// Mitsubishi GX Works2 project: 东芝分拣通信   PLC: Q10UDEH

TYPE ConveyorIO : STRUCT
  xUnloadCCW : BOOL;  (* 下料为反转 *)
  xUnloadAlarm : BOOL;  (* 下料报警 *)
  xUnload : BOOL;  (* 下料请求 *)
  xPutInto : BOOL;  (* 线体直接投入物料 *)
  xNotArriveAlarm : BOOL;  (* 未到达报警 *)
  xNextRun : BOOL;  (* 下段线体运行 *)
  xMotorCW : BOOL;  (* 电机正转 *)
  xMotorCCW : BOOL;  (* 电机反转 *)
  xManual : BOOL;  (* 手动 *)
  xloadCCW : BOOL;  (* 上料为反转 *)
  xLimitAlarrm : BOOL;  (* 限位报警 *)
  xLoad : BOOL;  (* 上料请求 *)
  xForward : BOOL;  (* 正转手动 *)
  xEmpty : BOOL;  (* 线体状态为空 *)
  xCWPresent : BOOL;  (* 正转检测有无传感器 *)
  xCCWPresent : BOOL;  (* 反转检测有无传感器 *)
  xBusy : BOOL;  (* 工作中 *)
  xBackward : BOOL;  (* 反转手动 *)
  xAuto : BOOL;  (* 自动 *)
  xPosLimit : BOOL;  (* 正限位 *)
  xNegLimit : BOOL;  (* 负限位 *)
  xOverWidthAlarm : BOOL;  (* 超宽报警 *)
  xError : BOOL;  (* 报警 *)
  iProductCategoryIn : INT;  (* 产品类型输入 *)
  iProductCategory : INT;  (* 产品类型记录 *)
  iProductCategoryOut : INT;  (* 产品类型输出 *)
  diDeviceID : DINT;  (* 设备编号 *)
  tUnloadAlarmDelay : TIME;  (* 下料报警时间设置 *)
  tLoadDelay : TIME;  (* 上料延时设置 *)
  xSizeDeficientDetect : BOOL;  (* 尺寸缺陷检测 *)
  xZoneClear : BOOL;  (* 初始化线体清除 *)
  tZoneClearTime : TIME;  (* 初始化线体清除时间 *)
  iTaskIDIn : INT;  (* 产品类型输入 *)
  iTaskID : INT;  (* 产品类型记录 *)
  iTaskIDOut : INT;  (* 产品类型输出 *)
  diDesConveyorIn : DINT;  (* 产品类型输入 *)
  diDesConveyor : DINT;  (* 产品类型记录 *)
  diDesConveyorOut : DINT;  (* 产品类型输出 *)
END_STRUCT END_TYPE

TYPE FanucRobotIO : STRUCT
  o_xColumn : ARRAY [0..3] OF BOOL;  (* 行号 *)
  o_xRow : ARRAY [0..3] OF BOOL;  (* 列号 *)
  o_xPutNumber : ARRAY [0..3] OF BOOL;  (* 放料位 *)
  o_xSortStart : BOOL;  (* 开始启动 *)
  i_xPutOver : BOOL;  (* 放货完成 *)
  i_xPickOver : BOOL;  (* 取货完成 *)
END_STRUCT END_TYPE

TYPE SortCommunicationIO : STRUCT
  i_iResponsPCPLC : INT;  (* 上位机写入-应答 *)
  i_iSortDoneAknPCPLC : INT;  (* 上位机写入-任务处理完成 *)
  i_arriBatteryStatus : ARRAY [1..128] OF INT;  (* 上位机写入-电池状态 *)
  o_iRequestPLCPC : INT;  (* 上位机读取-请求 *)
  o_iSortDonePLCPC : INT;  (* 上位机读取-分拣完成 *)
  i_iInfoWriteDone : INT;  (* 上位机写入-参数写入完成 *)
  i_xSortOver : BOOL;  (* 按钮，分拣完成 *)
  o_xSortDone : BOOL;  (* 状态，分拣完成 *)
END_STRUCT END_TYPE

// global labels: Global
VAR_GLOBAL
  g_xAuto AT M11 : BOOL;
  g_xManual : BOOL;
  g_xEStop AT X0 : BOOL;
  g_xReset : BOOL;
  g_xStackLampRed AT Y200 : BOOL;  (* 塔灯红 *)
  g_xStackLampAmber AT Y201 : BOOL;  (* 塔灯黄 *)
  g_xStackLampGreen AT Y202 : BOOL;  (* 塔灯绿 *)
  g_xBuzzer AT Y203 : BOOL;  (* 蜂鸣器 *)
  g_xStop AT X3 : BOOL;
  g_xAutoStart AT X2 : BOOL;  (* 启动按钮 *)
  g_xRemoteAutoStart AT M0 : BOOL;
  g_xRemoteAuto AT M10 : BOOL;
  g_iState AT D40 : INT;  (* 状态显示 *)
  g_iLocalAutoStep : BOOL;
  g_xAlarm : BOOL;
  g_xPause AT M3 : BOOL;  (* 暂停 *)
  g_diDeviceIDSelect AT D0 : DINT;
  g_xResetSingle AT M4 : BOOL;  (* 单线体复位 *)
  g_xInsertTask AT M5 : BOOL;  (* 插入任务 *)
  g_iInsertTaskID AT D2 : INT;  (* 插入任务号 *)
  g_iConveyorStatus AT D4 : INT;
  g_iInsertCategory AT D6 : INT;
  g_diInsertDesConveyor AT D8 : DINT;
  g_x20TcpFailed : BOOL;  (* 30预20通讯失败 *)
  g_xAutoLamp AT Y204 : BOOL;  (* 启动灯 *)
  g_iLoadTask AT D50 : ARRAY [0..13] OF INT;  (* 排队任务站，D50-D62 *)
  g_xAutoSwitch AT X1 : BOOL;  (* 手自动钥匙旋钮 *)
  g_xMute AT M2 : BOOL;  (* 静音按钮，报警消除时复位 *)
  g_xResetTask1 AT M9 : BOOL;  (* 复位排队任务按钮 *)
  g_xLoadPermit : ARRAY [1..2] OF BOOL;  (* 定位机排队任务允许 *)
  g_x40TcpFailed : BOOL;  (* 30预40通讯失败 *)
  g_xForceImport AT M1 : BOOL;  (* 强制入库 *)
  g_x24HourImport1Forbidden AT M12 : BOOL;  (* 24小时入库禁止1 *)
  g_x24HourImport2Forbidden AT M13 : BOOL;  (* 24小时入库禁止2 *)
  g_xPreChemImport1Forbidden AT M14 : BOOL;  (* 预化成入库禁止1 *)
  g_xPreChemImport2Forbidden AT M15 : BOOL;  (* 预化成入库禁止2 *)
  g_x24HourExport1Forbidden AT M16 : BOOL;  (* 24小时出库禁止 *)
  g_xPreChemExport1Forbidden AT M17 : BOOL;  (* 预化成出库禁止1 *)
  g_xPreChemExport2Forbidden AT M18 : BOOL;  (* 预化成出库禁止2 *)
  g_xPickDone : BOOL;  (* 分拣完成 *)
  g_xPickOver AT X4 : BOOL;  (* 注液机给我们的信号，待定 *)
END_VAR

// task Task_01 (event TRUE, interval 0, priority 31): POU_01

PROGRAM POU_01
VAR
  SortCommunication70210 : SortCommunication;  (* 分拣通信 *)
  Conveyor70210 : Conveyor;  (* 分拣线体 *)
  ConveyorIO70210 : ConveyorIO;  (* 分拣线体 *)
  RobotIO70210 : FanucRobotIO;  (* 分拣机器人 *)
  SortCommunicationIO70210 : SortCommunicationIO;  (* 分拣通信 *)
  ConveyorIO70211 : ConveyorIO;  (* 分拣线体的下一段线体，举个例子 *)
END_VAR
Conveyor70210(ConveyorMotor:=ConveyorIO70210);

SortCommunication70210(ConveyorIO:=ConveyorIO70210,SortCommunicationIO:= SortCommunicationIO70210 ,FanucRobotIO:= RobotIO70210);
SortCommunicationIO70210 .i_iResponsPCPLC:=D2705;
SortCommunicationIO70210 .i_iInfoWriteDone:=D2706;
SortCommunicationIO70210 .i_iSortDoneAknPCPLC:=D2707;
D3705:=SortCommunicationIO70210 .o_iRequestPLCPC;(*有料请求*)
D3706:=SortCommunicationIO70210 .o_iSortDonePLCPC;(*分拣完成信号*)
FOR Z0:=0 TO 127 BY 1 DO
	SortCommunicationIO70210 .i_arriBatteryStatus[Z0+1]:=D2708Z0;
END_FOR;

SortCommunicationIO70210.i_xSortOver:=X2;(*这个是手动放行按钮，可要可不要*)
RobotIO70210.i_xPickOver:=X0;(*机器人给的取货完成*)
RobotIO70210.i_xPutOver:=X1;(*机器人给的放货完成*)
Y0:=RobotIO70210.o_xSortStart;(*给机器人的开始启动*)
Y1:=RobotIO70210.o_xColumn[0];(*给机器人的行号*)
Y2:=RobotIO70210.o_xColumn[1];
Y3:=RobotIO70210.o_xColumn[2];
Y4:=RobotIO70210.o_xColumn[3];
Y5:=RobotIO70210.o_xRow[0];(*给机器人的列号*)
Y6:=RobotIO70210.o_xRow[1];
Y7:=RobotIO70210.o_xRow[2];
Y8:=RobotIO70210.o_xRow[3];
Y9:=RobotIO70210.o_xPutNumber[0];(*给机器人的放料位置*)
YA:=RobotIO70210.o_xPutNumber[1];
YB:=RobotIO70210.o_xPutNumber[2];
YC:=RobotIO70210.o_xPutNumber[3];

ConveyorIO70210.xUnload:=SortCommunicationIO70210.o_xSortDone AND ConveyorIO70211.xEmpty;(*比普通的下料多了个判断条件，需要分拣完成再下料*)
END_PROGRAM

FUNCTION_BLOCK SortCommunication
VAR
  m_iStep : INT;
END_VAR
VAR_IN_OUT
  ConveyorIO : ConveyorIO;
  SortCommunicationIO : SortCommunicationIO;
END_VAR
VAR
  m_iCoordinateX : INT;
  m_iCoordinateY : INT;
END_VAR
VAR_IN_OUT
  FanucRobotIO : FanucRobotIO;
END_VAR
VAR_OUTPUT
  o_iErrorNub : INT;
END_VAR
VAR
  ii : INT;
END_VAR
VAR CONSTANT
  ROW_NUB : INT := 8;  (* 每排的数量 *)
END_VAR
VAR
  m_xEno : BOOL;
END_VAR
(*********************************************************)
(*
DB1区(PC->PLC)100个字		
"字(16位）序号
(从1开始)"	功能描述	具体参数解释
1	应答	"1：复位
2：读码成功(参数写入完成)
101：条码空
102：条码规则校验失败
103：步号校验失败"
2	任务处理完成	"1：复位
2：处理完成"
3	"电芯状态，
128个电芯"	一个字代表两个电芯状态，1：合格，2,3,4:NG 

DB2区(PLC->PC)10个字		
"字(16位）序号
(从1开始)"	功能描述	具体参数解释
请求	"1：无板
2：请求分拣
"
分拣完成	"1：复位
2：挑选完成
3：撤销
"
跟机器人通信13个输出，2个输入
						13个输出分别是：4个表示行，4个表示列，4个表示不良信息，1个启动信号
						2个输入分别是：抓料完成，放料完成		

*)
(*********************************************************)
IF g_xAuto THEN
	(*——这里临时改一下，暂时人工挑选,所以需要分拣完成按钮——*)	
		IF LDP(TRUE,SortCommunicationIO.i_xSortOver)THEN
			m_iStep:=4;
		END_IF;(**)
(*——以上是暂时人工分拣的，以后删掉——*)
	CASE m_iStep OF
		0:(*//初始化*)
		SortCommunicationIO.o_iRequestPLCPC:=1;
		SortCommunicationIO.o_iSortDonePLCPC:=1;
		ii:=0;
		SortCommunicationIO.o_xSortDone:=0;
		m_iStep:=1;
		
		1:(*发送框码的扫码请求*)
		IF ConveyorIO.xEmpty THEN
			SortCommunicationIO.o_iRequestPLCPC:=1;
		ELSE
			SortCommunicationIO.o_iRequestPLCPC:=2;(*发2表示有料了，他就会扫码*)
		END_IF;
		(*//请求确认*)
		IF SortCommunicationIO.o_iRequestPLCPC=2 THEN(*加个条件，免得无脑跳Step2*)
			CASE SortCommunicationIO.i_iResponsPCPLC OF 
			0:;
			1:;(*//复位*)
			2:(*//读码（入库申请）成功*)
				m_iStep:=2;
				ii:=0;
				m_iCoordinateX:=1;(*//框码扫码成功后把坐标改为1,1*)
				m_iCoordinateY:=1;
			3:(*//取放货完成*)
				ConveyorIO.xPutInto:=1; 
			4:(*//旋转*)
				;
			5:(*//不旋转*)
				;
			101:(*//条码空*)
				o_iErrorNub:=101;
			102:(*//条码规则检验失败*)
				o_iErrorNub:=102;
			103:(*//步号校验失败*)
				o_iErrorNub:=103;
			104:(*//无库位可用*)
				o_iErrorNub:=104;
			END_CASE;
		END_IF;	
		
		2:(*//料框位置抓取*)		
		IF ii=129 THEN(*129表示所有有问题的都抓完了*)
			m_iStep:=4;
		ELSE(*有不良品*)
			FanucRobotIO.o_xSortStart:=1;(*//从料框取料*)
			FanucRobotIO.o_xColumn[3]:=m_iCoordinateX/8=1;(*XY的偏移量计算在末尾*)
			FanucRobotIO.o_xColumn[2]:=(m_iCoordinateX MOD 8)/4=1;
			FanucRobotIO.o_xColumn[1]:=(m_iCoordinateX MOD 4)/2=1;
			FanucRobotIO.o_xColumn[0]:=(m_iCoordinateX MOD 2)/1=1;
			FanucRobotIO.o_xRow[3]:=m_iCoordinateY/8=1;			
			FanucRobotIO.o_xRow[2]:=(m_iCoordinateY MOD 8)/4=1;
			FanucRobotIO.o_xRow[1]:=(m_iCoordinateY MOD 4)/2=1;
			FanucRobotIO.o_xRow[0]:=(m_iCoordinateY MOD 2)/1=1;
			CASE SortCommunicationIO.i_arriBatteryStatus[ii] OF
			1:(*合格*)
					;
			2:(*容量不足*)
					FanucRobotIO.o_xPutNumber[0]:=1;	
			3:(*电压不足*)
					FanucRobotIO.o_xPutNumber[1]:=1;	
			4:(*阻值错误*)
					FanucRobotIO.o_xPutNumber[2]:=1;	
			5:(*电压过高*)
					FanucRobotIO.o_xPutNumber[3]:=1;	
			END_CASE;
		END_IF;
		IF LDP(TRUE,FanucRobotIO.i_xPickOver) THEN(*//抓取动作完成*)
			m_iStep:=3;
		END_IF;
	
		3:(*//放入下料皮带线*)
			FanucRobotIO.o_xSortStart:=0;(*//从料框取料*)
			FanucRobotIO.o_xColumn[3]:=0;(*XY的偏移量计算在末尾*)
			FanucRobotIO.o_xColumn[2]:=0;
			FanucRobotIO.o_xColumn[1]:=0;
			FanucRobotIO.o_xColumn[0]:=0;
			FanucRobotIO.o_xRow[3]:=0;
			FanucRobotIO.o_xRow[2]:=0;
			FanucRobotIO.o_xRow[1]:=0;
			FanucRobotIO.o_xRow[0]:=0;
		IF LDP(TRUE,FanucRobotIO.i_xPutOver) THEN(*//抓取动作完成*)
		(*这个得放货完成在复位，方便step2给*)
		FanucRobotIO.o_xPutNumber[0]:=0;
		FanucRobotIO.o_xPutNumber[1]:=0;
		FanucRobotIO.o_xPutNumber[2]:=0;
		FanucRobotIO.o_xPutNumber[3]:=0;
			m_iStep:=2;
		END_IF;	
		
		4:
		IF  NOT SortCommunicationIO.o_xSortDone  THEN(*这里表示只给一下2*)
				SortCommunicationIO.o_iSortDonePLCPC:=2;
				SortCommunicationIO.o_xSortDone:=1;
		END_IF;		
		IF SortCommunicationIO.i_iSortDoneAknPCPLC =2 THEN
			SortCommunicationIO.o_iSortDonePLCPC:=1;
			m_iCoordinateX:=1;
			m_iCoordinateY:=1;
		END_IF;	
			IF ConveyorIO.xEmpty THEN
				m_iStep:=0;
			END_IF;
	END_CASE;
	IF LDP(TRUE,m_iStep=2 AND SortCommunicationIO.i_iInfoWriteDone=2) THEN(*判断哪个地方是有问题的*)
		FOR ii:=ii+1 TO 128 BY 1 DO
			IF SortCommunicationIO.i_arriBatteryStatus[ii]<>1 THEN
				m_iCoordinateX:=((ii-1) MOD ROW_NUB);
				m_iCoordinateY:=(ii-1)/ROW_NUB+1;(*把上位机给的编号值对应到二维的偏移上*)
				EXIT;
			END_IF;
		END_FOR;
	END_IF;
END_IF;(*g_xauto*)	
IF  g_diDeviceIDSelect=ConveyorIO.diDeviceID AND g_xResetSingle THEN(*复位线体时，同时复位步数和请求，重新来一遍*)
	m_iStep:=0;
END_IF;	
IF  NOT g_xAuto THEN
		SortCommunicationIO.o_iRequestPLCPC:=0;
		SortCommunicationIO.o_iSortDonePLCPC:=0;
END_IF;
END_FUNCTION_BLOCK

FUNCTION_BLOCK Conveyor
VAR
  m_xPresentDelay : BOOL;  (* 有无判断延时 *)
  m_xLoadDelayOut : BOOL;  (* 上料延时输出 *)
  m_xInitial : BOOL;  (* 初始化 *)
  m_tUnloadTimer : TIME;  (* 下料计时器 *)
  m_tPresentDelayCurrentTime : TIME;
  m_tonUnloadAlam : TON;  (* 下料报警定时器 *)
  m_tonPresentDelay : TON;  (* 物料有无判断延时，防止误动作 *)
  m_tonNotArriveAlarm : TON;  (* 未到达报警计时 *)
  m_tonLoadDelay : TON;  (* 上料延时 *)
  m_tNotArriveCurrentTime : TIME;  (* 未到达报警计时当前时间 *)
  m_tLoadTimer : TIME;  (* 上料计时器 *)
  iStep : INT;  (* 上料步骤 *)
  m_wStateWord : INT;
END_VAR
VAR_IN_OUT
  ConveyorMotor : ConveyorIO;  (* 输送线输入输出 *)
END_VAR
VAR
  m_tonZoneClear : TON;  (* 初始化清除 *)
  m_tZoneClearCurrentTime : TIME;  (* 初始化清除当前时间 *)
  m_xAutoClear : BOOL;  (* 初始化清除标志位 *)
  m_xZoneClearDone : BOOL;  (* 初始化清除完成 *)
END_VAR
(*////////////////////////////////////////////////////////////////////////////////////////////////////////////
//传输线控制FB块，可控制单方向线体，双向旋转线体，支持双向上下料            
//线体初始化后为空的情况下输入xLoad信号即可进行上料动作，使用xLoadCCW信号可反方向上料
//增加了产品信息和产品种类的储存，当传输线为空和上料进行标志位为零的情况下清除产品信息和产品种类
//使用方式是在置位xLoad信号后，把产品信息和产品种类传入，等下料后自动清零
//线体不为空的情况下使用xUnload信号可进行下料动作，物料有无传感器的下降沿后出发计时器，延时断开传输线旋转
//单方向传输线体把xLoadCCW、xUnloadCCW设置为零，双向线体上料方向和下料反向的,方向固定的 把xUnloadCCW设置为1
//双方向线体双向都能上下料的要根据上料的方向来设置xLoadCCW,xUnloadCCW
//增加工作中信号xBusy当电机正转 显示为工作中
//增加上下料超时报警，xLoadAlarm，xUnloadAlarm，设定时间在LOAD_UNLOAD_TIME常量上，现在设置的为30秒
//增加xPutInto信号，用于直接投入的物料，检测开关感应到后，直接进入下料流程，上升沿有效
//离开延时改为变量 iLeaveDelay 默认为0 离开检测开关离输送线尾端比较远的线体需要根据情况设定100ms为单位
//增加初始化标志位，增加进入延时时间，初始化为进入延时时间为0 ，离开延时时间为2S，通过外围接口可以更改
//修改信息  修改后请增加版本
//12-17进行了优化，增加了未到达报警，当物料未传送到下一设备，就报未到达报警，使用xNextRun标志位制作，没有正常到达
//第0步，不能跳转到第一步把标志位复位，即出现中断情况，2秒后报警
//修改信息  修改后请增加版本
//上料延时增加为50ms防止干扰信号
//nextrun信号在 第三步也要复位
//增加限位报警
//增加超宽报警
//增加产品型号输出在下料的时候把产品型号输送给下一段线体
//增加线体单独复位
//增加任务插入功能配合全局变量
//增加暂停功能
//增加线体状态字显示  0 空闲 1：有料  2 工作中  3  超限报警 4 超宽报警  5 未到达报警  6 下料超时报警
//空料判断放在自动前，进行有无报警判断，然后跳转
//修改超限报警，与尺寸检测报警
////YAO      V1.0
//把所有的IF语句去掉，  IF语句占用指针存储区，容易造成存储区不足的现象
////YAO      V1.1
//初始化清除线体标志位xZoneClear
//ZPA zero pressure accumulation  Term that describes the Conveyor controls and mechanical scheme that will 
//cause loads to queue on a conveyor in discrete zones such that loads do not touch each other(wrapped boxed tray tote carton)
//除了产品信息外，还增加了目标地址，任务类型的数据传递。
//YAO      V1.0
///////////////////////////////////////////////////////////////////////////////////////////////////////////
(*********************************************************)
(*//初始化，
//上料延时位0S，下料报警延时为30S
//下料延时设一个比较大的时间，主要依靠xunload标志位来停止输送线，特殊情况可以用延时来停止物流线下料
//设置时间大的时候计时器会失效*)
IF NOT m_xInitial THEN
	ConveyorMotor.tLoadDelay:=T#100ms;
	ConveyorMotor.tUnloadAlarmDelay:=T#30s;
	ConveyorMotor.xPosLimit:=1;
	ConveyorMotor.xNegLimit:=1;
	ConveyorMotor.xSizeDeficientDetect:=0;
	ConveyorMotor.xZoneClear:=0;
	ConveyorMotor.tZoneClearTime:=T#10s;
	m_xInitial:=1;
END_IF;
(*//自动
//复位信号把步号置0，但xLoad与xUnload没有复位，调用程序需要注意复位后把这两个信号置零，以免发生误动作
//物料有无判断增加延时，防止开自动瞬间误动作发生*)
m_tonPresentDelay(IN:= ConveyorMotor.xCWPresent OR ConveyorMotor.xCCWPresent,
					PT:=T#100ms,
					Q:= m_xPresentDelay,
					ET:= m_tPresentDelayCurrentTime);
CASE iStep OF
0:(*//初始化*)
	ConveyorMotor.xMotorCW:=0;
	ConveyorMotor.xMotorCCW:=0;
	ConveyorMotor.xNextRun:=0;
	ConveyorMotor.iProductCategoryOut:=0;
	ConveyorMotor.iTaskIDOut:=0;
	ConveyorMotor.diDesConveyorOut:=0;
	out(NOT m_xPresentDelay,ConveyorMotor.xEmpty);(*	//判断物料有无传感器*)	
	mov(m_xPresentDelay AND g_xAuto AND NOT ConveyorMotor.xError,3,iStep);(*//自动情况下进行跳转*)(*无超限报警*)
	mov(NOT m_xPresentDelay AND g_xAuto AND NOT ConveyorMotor.xError,1,iStep);
1: (*//上料*)
	rst(ConveyorMotor.xLoad ,ConveyorMotor.iProductCategory);(*//上料开始清除产品信息*)
	rst(ConveyorMotor.xLoad ,ConveyorMotor.iTaskID);
	rst(ConveyorMotor.xLoad ,ConveyorMotor.diDesConveyor);
	mov(ConveyorMotor.xLoad,2,iStep);
2: (*//上料完成*)
	ConveyorMotor.iProductCategory:=ConveyorMotor.iProductCategoryIn;(* //产品信息传入*)
	ConveyorMotor.iTaskID:=ConveyorMotor.iTaskIDIn;
	ConveyorMotor.diDesConveyor:=ConveyorMotor.diDesConveyorIn;
	set(ConveyorMotor.xloadCCW,ConveyorMotor.xMotorCCW);
	rst(ConveyorMotor.xloadCCW,ConveyorMotor.xMotorCW);
	set(NOT ConveyorMotor.xloadCCW,ConveyorMotor.xMotorCW);
	rst(NOT ConveyorMotor.xloadCCW,ConveyorMotor.xMotorCCW);	
	m_tonLoadDelay(IN:= (ConveyorMotor.xCWPresent AND NOT ConveyorMotor.xloadCCW) 
												OR (ConveyorMotor.xCCWPresent AND ConveyorMotor.xloadCCW) ,
										PT:= ConveyorMotor.tLoadDelay ,
										Q:= m_xLoadDelayOut ,
										ET:= m_tLoadTimer );
	mov(m_xLoadDelayOut,3, iStep);
3:(*//下料请求*)	
	ConveyorMotor.xMotorCW:=0;
	ConveyorMotor.xMotorCCW:=0;
	ConveyorMotor.xEmpty:=0;
	mov(ConveyorMotor.xUnload AND NOT ConveyorMotor.xOverWidthAlarm,4,iStep);
4:(*	//下料完成*)
	set(ConveyorMotor.xUnloadCCW,ConveyorMotor.xMotorCCW);
	rst(ConveyorMotor.xUnloadCCW,ConveyorMotor.xMotorCW);
	set(NOT ConveyorMotor.xUnloadCCW,ConveyorMotor.xMotorCW);
	rst(NOT ConveyorMotor.xUnloadCCW,ConveyorMotor.xMotorCCW);	
	ConveyorMotor.xNextRun:=1; (*下一段线体旋转*)
	ConveyorMotor.iProductCategoryOut:=ConveyorMotor.iProductCategory;(*产品型号输出给下一段线体*)
	ConveyorMotor.iTaskIDOut:=ConveyorMotor.iTaskID;
	ConveyorMotor.diDesConveyorOut:=ConveyorMotor.diDesConveyor;
	mov( NOT ConveyorMotor.xUnload , 0, istep );
END_CASE;
(*In-feed zone clear and ready to accept a load from Upstream Conveyor*)
set(ldp(TRUE,g_xAuto) ,m_xAutoClear);
rst(ldf(TRUE,g_xAuto) ,m_xAutoClear);
m_tonZoneClear(IN:= m_xAutoClear AND ConveyorMotor.xZoneClear ,PT:= ConveyorMotor.tZoneClearTime ,Q:=m_xZoneClearDone ,ET:= m_tZoneClearCurrentTime );
set(m_xAutoClear AND ConveyorMotor.xZoneClear,ConveyorMotor.xMotorCW);
mov( m_xAutoClear AND ConveyorMotor.xZoneClear, 0 ,iStep );
rst(  ldf(TRUE, m_xAutoClear ) ,ConveyorMotor.xMotorCW);
rst( m_xZoneClearDone OR m_xPresentDelay  , m_xAutoClear );
(*投入上料，搬出下料，也可用来初始化*)
movp( ConveyorMotor.xPutInto, 0 , iStep );
(*//当前任务显示*)
movp( ConveyorMotor.diDeviceID=g_diDeviceIDSelect , ConveyorMotor.iProductCategory , g_iInsertCategory );
movp( ConveyorMotor.diDeviceID=g_diDeviceIDSelect , ConveyorMotor.iTaskID , g_iInsertTaskID );
dmovp( ConveyorMotor.diDeviceID=g_diDeviceIDSelect , ConveyorMotor.diDesConveyor , g_diInsertDesConveyor );
(*//插入任务*)
mov(g_xInsertTask AND ConveyorMotor.diDeviceID=g_diDeviceIDSelect ,g_iInsertCategory , ConveyorMotor.iProductCategory );
mov(g_xInsertTask AND ConveyorMotor.diDeviceID=g_diDeviceIDSelect , g_iInsertTaskID , ConveyorMotor.iTaskID );
dmov(g_xInsertTask AND ConveyorMotor.diDeviceID=g_diDeviceIDSelect , g_diInsertDesConveyor , ConveyorMotor.diDesConveyor );
(*//单线体复位，当设备号与本线体一致的时候执行复位*)
mov(g_xResetSingle AND ConveyorMotor.diDeviceID=g_diDeviceIDSelect , 0 , iStep );
rst(g_xResetSingle AND ConveyorMotor.diDeviceID=g_diDeviceIDSelect ,ConveyorMotor.xNextRun );
rst(g_xResetSingle AND ConveyorMotor.diDeviceID=g_diDeviceIDSelect  ,ConveyorMotor.xLimitAlarrm );
rst(g_xResetSingle AND ConveyorMotor.diDeviceID=g_diDeviceIDSelect  ,ConveyorMotor.xOverWidthAlarm );
(*//手动*)
(*//正转*)
set( g_xManual 
AND ConveyorMotor.xForward 
AND ConveyorMotor.xBackward=0 
AND ConveyorMotor.xMotorCCW=0 
AND g_xEStop  , 
ConveyorMotor.xMotorCW);
rst((g_xManual 
AND (NOT ConveyorMotor.xForward  
OR ConveyorMotor.xBackward 
OR ConveyorMotor.xMotorCCW )) 
OR NOT g_xEStop,
ConveyorMotor.xMotorCW);
(*//反转*)		
set(g_xManual 
AND ConveyorMotor.xBackward 
AND ConveyorMotor.xForward=0 
AND ConveyorMotor.xMotorCW=0 
AND g_xEStop ,
ConveyorMotor.xMotorCCW);
rst((g_xManual AND 
(NOT ConveyorMotor.xBackward  
OR ConveyorMotor.xForward 
OR ConveyorMotor.xMotorCW ) ) 
OR NOT g_xEStop,
ConveyorMotor.xMotorCCW);
mov(g_xManual ,0,iStep);(*//手动后上下料程序步骤清零*)
(*暂停*)
rst(g_xPause,ConveyorMotor.xMotorCCW);
rst( g_xPause , ConveyorMotor.xMotorCW );
rst(NOT g_xAuto AND NOT g_xManual,ConveyorMotor.xMotorCCW);
rst( NOT g_xAuto AND NOT g_xManual, ConveyorMotor.xMotorCW );
(*工作中信号输出*)
ConveyorMotor.xBusy:=ConveyorMotor.xMotorCCW OR ConveyorMotor.xMotorCW;
(*//未到达报警*)
m_tonNotArriveAlarm(IN:= iStep=0 AND ConveyorMotor.xNextRun  ,PT:= T#2s,Q:= ConveyorMotor.xNotArriveAlarm ,ET:= m_tNotArriveCurrentTime );
(*//下料超时报警*)
m_tonUnloadAlam(IN:= iStep=4,PT:=ConveyorMotor.tUnloadAlarmDelay,Q:= ConveyorMotor.xUnloadAlarm,ET:=m_tUnloadTimer );
(*//限位报警,进料检测开关失效*)
set(  ( ((ConveyorMotor.xloadCCW AND NOT ConveyorMotor.xNegLimit)            (*反转上料，碰到负限位*)
			OR  ( NOT ConveyorMotor.xloadCCW AND NOT ConveyorMotor.xPosLimit)) (*正转上料，碰到正限位*)
		AND iStep=2) (*上料过程*)
	OR
	( iStep=4 (*下料过程*)
		AND( (ConveyorMotor.xUnloadCCW AND NOT ConveyorMotor.xPosLimit)  
			OR (NOT ConveyorMotor.xUnloadCCW AND NOT ConveyorMotor.xNegLimit)))  ,  
	ConveyorMotor.xLimitAlarrm );
mov( ( ((ConveyorMotor.xloadCCW AND NOT ConveyorMotor.xNegLimit)            (*反转上料，碰到负限位*)
			OR  ( NOT ConveyorMotor.xloadCCW AND NOT ConveyorMotor.xPosLimit)) (*正转上料，碰到正限位*)
		AND iStep=2) (*上料过程*)
	OR
	( iStep=4 (*下料过程*)
		AND( (ConveyorMotor.xUnloadCCW AND NOT ConveyorMotor.xPosLimit)  
			OR (NOT ConveyorMotor.xUnloadCCW AND NOT ConveyorMotor.xNegLimit)))  ,
	0,
	iStep);
(*//超宽报警*)
set( (iStep=3 OR iStep=1) AND (NOT ConveyorMotor.xNegLimit OR NOT ConveyorMotor.xPosLimit) , ConveyorMotor.xOverWidthAlarm  );
(*//尺寸不足报警*)
(*//有料状态下检测两个开关都要有信号*)
set( iStep=3 AND ConveyorMotor.xSizeDeficientDetect AND (NOT ConveyorMotor.xCCWPresent OR NOT ConveyorMotor.xCWPresent) ,  ConveyorMotor.xOverWidthAlarm );
mov( iStep=3 AND ConveyorMotor.xSizeDeficientDetect AND (NOT ConveyorMotor.xCCWPresent OR NOT ConveyorMotor.xCWPresent),0,iStep);
(*//总报警*)
ConveyorMotor.xError:=ConveyorMotor.xLimitAlarrm
					OR ConveyorMotor.xNotArriveAlarm
					OR ConveyorMotor.xUnloadAlarm                                             
					OR ConveyorMotor.xOverWidthAlarm;

(*//状态输出*)(*状态显示，容易造成指针容量不足*)
mov( ConveyorMotor.xEmpty AND NOT ConveyorMotor.xBusy , 0 , m_wStateWord);
mov( ConveyorMotor.xEmpty=0 , 							1 , m_wStateWord);
mov( ConveyorMotor.xBusy , 								2 , m_wStateWord);
mov( ConveyorMotor.xLimitAlarrm , 						3, 	m_wStateWord);
mov(ConveyorMotor.xOverWidthAlarm , 					4 , m_wStateWord);
mov( ConveyorMotor.xNotArriveAlarm , 					5 , m_wStateWord);
mov( ConveyorMotor.xUnloadAlarm, 						6 , m_wStateWord);
(*选择本线体后，将状态赋值给全局变量进行显示*)
mov( ConveyorMotor.diDeviceID=g_diDeviceIDSelect , m_wStateWord, g_iConveyorStatus );
END_FUNCTION_BLOCK

FUNCTION_BLOCK FanucRobot
VAR_IN_OUT
  FanucRobotIO : FanucRobotIO;
END_VAR
VAR
  m_iSNO : INT;
  m_xPNSPass : BOOL;  (* 收到程序号 *)
  m_tonStartDelay : TON;  (* 启动延时 *)
  m_xStartDelay : BOOL;
  m_tStartDelayCurrentTime : TIME;
END_VAR
(***********************************************************
发那科机器人自动启动程序


***********************************************************)

(*无自动状态，示教盒处于本地状态，把各标志位复位*)
IF FanucRobotIO.i_xTPENBL AND NOT g_xAuto THEN
	FanucRobotIO.o_xPNSTROBE:=0;
	FanucRobotIO.o_xCSTOPI:=0;
	FanucRobotIO.o_xPROD_START:=0;
	FanucRobotIO.o_xRESET:=0;
END_IF;
(*远程模式*)
IF g_xAuto THEN
	FanucRobotIO.o_xREMOTE:=1;
	ELSE
	FanucRobotIO.o_xREMOTE:=0;
END_IF;
(*程序启动后复位启动标志位*)
(*//IF FanucRobotIO.i_xPROG_RUN AND FanucRobotIO.i_xBUSY THEN
//	FanucRobotIO.i_xCommandStart:=0;
//END_IF;*)
(*示教盒旋清除报警*)
IF ldf(TRUE,FanucRobotIO.i_xTPENBL)THEN
	FanucRobotIO.o_xRESET:=1;
	FanucRobotIO.o_xCSTOPI:=1;
END_IF;
(*启动程序号条件*)
IF FanucRobotIO.i_xSYSRDY 
	AND FanucRobotIO.i_xCMDENBL
(*//	AND FanucRobotIO.i_xCommandStart*)
	AND NOT FanucRobotIO.i_xPROG_RUN 
	AND NOT FanucRobotIO.i_xBUSY THEN
	FanucRobotIO.o_xRESET:=0;
	FanucRobotIO.o_xCSTOPI:=0;
	IF FanucRobotIO.i_iMotionNumber <> 0 (*只要动作编号不为0，就给他信号*)
		AND NOT FanucRobotIO.o_xPNSTROBE THEN
		FanucRobotIO.o_xPNSTROBE:=1;
		FanucRobotIO.o_xPROD_START:=1;
		FanucRobotIO.o_iPNS:=FanucRobotIO.i_iMotionNumber;(*并把任务号传给他*)
	END_IF;
	(*程序号校验*)
	IF FanucRobotIO.i_xSNACK THEN(*数据传回之后再校验*)
		m_iSNO:=BITARR_TO_INT(FanucRobotIO.i_arrxSNO[0] , 8 );
		IF m_iSNO=FanucRobotIO.o_iPNS THEN
			m_xPNSPass:=1;(*校验成功,等100MS复位Start信号*)
			FanucRobotIO.o_xPNSTROBE:=0;
		ELSE
			FanucRobotIO.o_xPNSFailed:=1;(*校验失败*)
			FanucRobotIO.o_xPROD_START:=0;(*立刻复位，不生成任务*)
		END_IF;
	END_IF;
END_IF;
m_tonStartDelay(IN:= m_xPNSPass ,PT:= T#100ms ,Q:= m_xStartDelay ,ET:=m_tStartDelayCurrentTime );
IF m_xStartDelay THEN
	FanucRobotIO.o_xPROD_START:=0;
(*//	FanucRobotIO.i_xCommandStart:=0;*)
	m_xPNSPass:=0;
END_IF;
END_FUNCTION_BLOCK
